PROGRAM Axis05_Manual
VAR
//System_Bit
	Always_ON	:	BOOL	:=TRUE	;//상시 ON 
	Always_OFF	:	BOOL	:=FALSE	;//상시 OFF
END_VAR
VAR // added by the converter: edge detectors and wires of the graphical bodies
    _rt1, _rt2, _rt3 : R_TRIG;
END_VAR

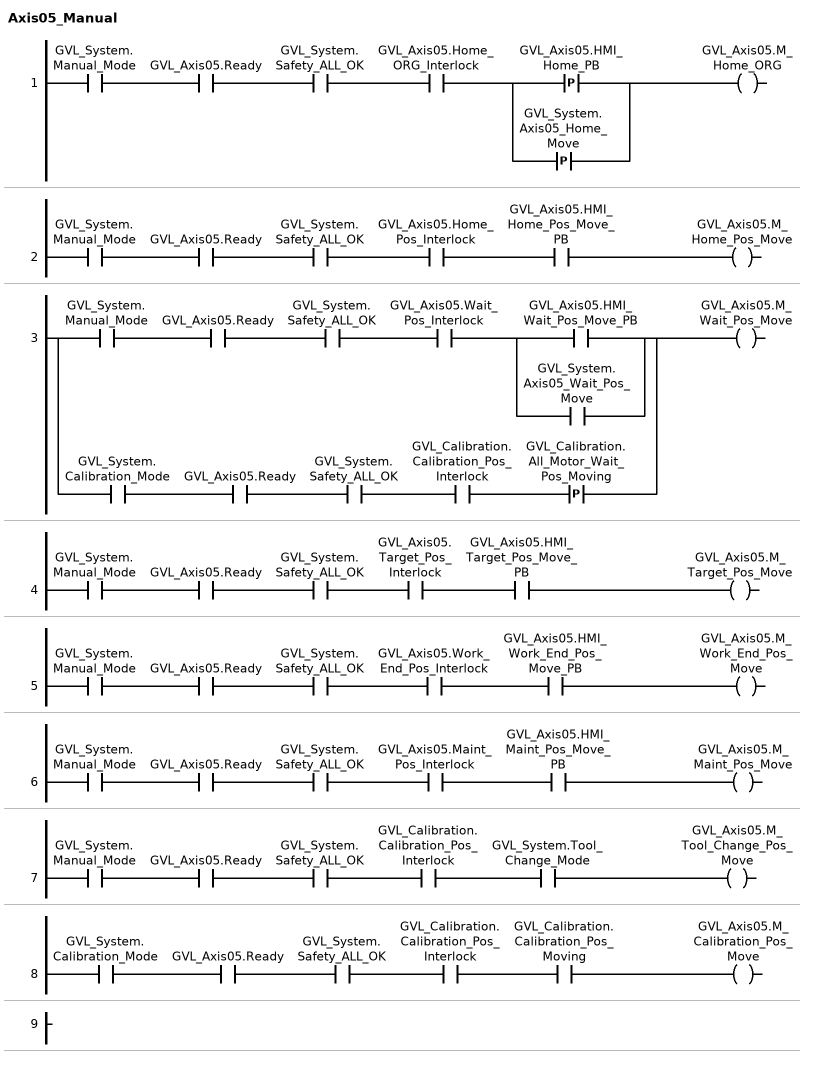
// NETWORK 1
_rt1(CLK := GVL_Axis05.HMI_Home_PB);
_rt2(CLK := GVL_System.Axis05_Home_Move);
GVL_Axis05.M_Home_ORG := GVL_System.Manual_Mode AND GVL_Axis05.Ready AND GVL_System.Safety_ALL_OK AND GVL_Axis05.Home_ORG_Interlock AND (_rt1.Q OR _rt2.Q);

// NETWORK 2
GVL_Axis05.M_Home_Pos_Move := GVL_System.Manual_Mode AND GVL_Axis05.Ready AND GVL_System.Safety_ALL_OK AND GVL_Axis05.Home_Pos_Interlock AND GVL_Axis05.HMI_Home_Pos_Move_PB;

// NETWORK 3
_rt3(CLK := GVL_Calibration.All_Motor_Wait_Pos_Moving);
GVL_Axis05.M_Wait_Pos_Move := GVL_System.Manual_Mode AND GVL_Axis05.Ready AND GVL_System.Safety_ALL_OK AND GVL_Axis05.Wait_Pos_Interlock AND (GVL_Axis05.HMI_Wait_Pos_Move_PB OR GVL_System.Axis05_Wait_Pos_Move) OR GVL_System.Calibration_Mode AND GVL_Axis05.Ready AND GVL_System.Safety_ALL_OK AND GVL_Calibration.Calibration_Pos_Interlock AND _rt3.Q;

// NETWORK 4
GVL_Axis05.M_Target_Pos_Move := GVL_System.Manual_Mode AND GVL_Axis05.Ready AND GVL_System.Safety_ALL_OK AND GVL_Axis05.Target_Pos_Interlock AND GVL_Axis05.HMI_Target_Pos_Move_PB;

// NETWORK 5
GVL_Axis05.M_Work_End_Pos_Move := GVL_System.Manual_Mode AND GVL_Axis05.Ready AND GVL_System.Safety_ALL_OK AND GVL_Axis05.Work_End_Pos_Interlock AND GVL_Axis05.HMI_Work_End_Pos_Move_PB;

// NETWORK 6
GVL_Axis05.M_Maint_Pos_Move := GVL_System.Manual_Mode AND GVL_Axis05.Ready AND GVL_System.Safety_ALL_OK AND GVL_Axis05.Maint_Pos_Interlock AND GVL_Axis05.HMI_Maint_Pos_Move_PB;

// NETWORK 7
GVL_Axis05.M_Tool_Change_Pos_Move := GVL_System.Manual_Mode AND GVL_Axis05.Ready AND GVL_System.Safety_ALL_OK AND GVL_Calibration.Calibration_Pos_Interlock AND GVL_System.Tool_Change_Mode;

// NETWORK 8
GVL_Axis05.M_Calibration_Pos_Move := GVL_System.Calibration_Mode AND GVL_Axis05.Ready AND GVL_System.Safety_ALL_OK AND GVL_Calibration.Calibration_Pos_Interlock AND GVL_Calibration.Calibration_Pos_Moving;

// NETWORK 9

END_PROGRAM

(* stored: Version 1.1.0.1, ProductVersion 3.1.4024.15
   POU Axis05_Manual: Id {9e769e66-efb3-499d-8b36-05e79ce2e9bc}, SpecialFunc None *)
